// TIA Portal V17 export
// export: Created 2024-09-02T12:50:09.6307871Z, ExportSetting WithDefaults, DisplayName Totally Integrated Automation Portal, DisplayVersion V17, DisplayName TIA Portal Openness, DisplayVersion V17, DisplayName TIA Portal Version Control Interface, DisplayVersion V17, DisplayName STEP 7 Professional, DisplayVersion V17, DisplayName STEP 7 Safety, DisplayVersion V17, DisplayName WinCC Professional, DisplayVersion V17
DATA_BLOCK "GraDB2_FG02_Station_OP70"   // DB1362
{ S7_Optimized_Access := 'TRUE'; DB_Accessible_From_OPC_UA := 'FALSE' }
AUTHOR : VAF
FAMILY : SK
NAME : SK
VERSION : 0.1
// stored: AutoNumber false, DBAccessibleFromOPCUA false, IsOnlyStoredInLoadMemory false, IsRetainMemResEnabled false, IsWriteProtectedInAS false, MemoryReserve 0
   VAR
      Home { ExternalWritable := 'False'} : Bool;   // Grundstellung
      Home_Mechanic { ExternalWritable := 'False'} : Bool;   // Grundstellung Mechanik / Basic position mechanic
      Home_SQ { ExternalWritable := 'False'} : Bool;   // Grundstellung Schrittkette / Basic position Step chain
      Finished_Screwdriver { ExternalWritable := 'False'} : Bool := false;   // Fertigmeldung / Finished message
      Finished_OK_Screwdriver : Bool;
      Finished_NOK_Screwdriver : Bool;
      Finished_Reset_Screwdriver { ExternalWritable := 'False'} : Bool;   // Fertigmeldung Reset / Finished Reset
      SQ_Finished_Screwdriver { ExternalWritable := 'False'} : Bool;   // Ablauf Schrittkette fertig / Sequence cycle finished
      Finished_Camera { ExternalWritable := 'False'} : Bool := false;   // Fertigmeldung / Finished message
      Finished_OK_Camera : Bool;
      Finished_NOK_Camera : Bool;
      Finished_Reset_Camera { ExternalWritable := 'False'} : Bool;   // Fertigmeldung Reset / Finished Reset
      SQ_Finished_Camera { ExternalWritable := 'False'} : Bool;   // Ablauf Schrittkette fertig / Sequence cycle finished
      Workers { ExternalWritable := 'False'; S7_SetPoint := 'True'} : "TypeSKS_OPERATOR";   // Schrittmerker / Step marker
      "MM140 Y- Axis Gripper" { S7_SetPoint := 'True'} : "TypeSKS_HORI";
      "MM150 Z- Axis Gripper" { S7_SetPoint := 'True'} : "TypeSKS_VERT";
      Gripper { S7_SetPoint := 'True'} : "TypeSKS_GRIP";
      "MM160 Z- Axis Screwdriver" { S7_SetPoint := 'True'} : "TypeSKS_VERT";
      "MM170 Z- Axis Screwdriver unit" { S7_SetPoint := 'True'} : "TypeSKS_VERT";
      "MM180 Z- Axis Screwdriver unit Clamp" { S7_SetPoint := 'True'} : "TypeSKS_STP";
      "MM190 Z- Axis Screwdriver unit Clamp" { S7_SetPoint := 'True'} : "TypeSKS_STP";
      ScrewDriver { S7_SetPoint := 'True'} : "TypeSKS_Desutter";
      Camera { S7_SetPoint := 'True'} : "TypeSKS_Omron";
      Feeder_Screw : Struct
         "A" : Struct
            on : Bool;
            off : Bool;
            Part_Out : Bool;
         END_STRUCT;
         H : Struct
            on : Bool;
            off : Bool;
            R_Part_insite : Bool;
            R_Part_in_Undefined_position : Bool;
            R_Part_in_pipe : Bool;
            S_Part_insite : Bool;
            S_Part_in_Undefined_position : Bool;
            S_Part_in_pipe : Bool;
         END_STRUCT;
         Status : Struct
            Part_Inside : Bool;
            Part_in_Undefined_Position : Bool;
            Part_in_Undefined_Position_Alarm_Active : Bool;
         END_STRUCT;
      END_STRUCT;
      Part_in_Gripper_Controle : Struct
         Fallen : Bool;
         Part_in_picking_Pos_Confirm : Bool;
      END_STRUCT;
      NIO_Controle : Struct
         HMI_Input : Struct
            X1 : Int;
            X2 : Int;
            Restart : Bool;
         END_STRUCT;
         Staus : Struct
            Warning : Bool;
            Error : Bool;
         END_STRUCT;
         Actual : Struct
            Counter_NOK : IEC_COUNTER;
         END_STRUCT;
      END_STRUCT;
      Retry : Array[1..8] of Struct
         Max_Retry : Int;
         Actual_Retry : Int;
         "Counter" : IEC_COUNTER;
      END_STRUCT;
      "Station Finished_Screwdriver" : Bool;
      fpDamperCap_Cam_Deselection : Bool;
      fnDamperCap_Cam_Deselection : Bool;
   END_VAR
BEGIN
   Retry[1..8].Max_Retry := 2;
END_DATA_BLOCK
